{attribute addProperty BoxType "EK1122-0000-0018"}
{attribute addProperty Id "Beckhoff_EJ3xxxsub_EK1100EK1100_179A0949162"}
{attribute addProperty CRC "1763837838"}
{attribute addProperty SizeInBites "16"}
{attribute addProperty SizeInBytes "2"}
TYPE Beckhoff_EJ3xxxEK1122_6922078E EXTENDS EK1122_179A0949 :
STRUCT
	{attribute addProperty Name "Beckhoff_EJ3xxxsub_EK1100"}
	Beckhoff_EJ3xxxsub_EK1100 : EK1100_179A0949;
END_STRUCT
END_TYPE

(* stored: Version 1.2.0.0, ProductVersion 3.1.4024.9
   DUT Beckhoff_EJ3xxxEK1122_6922078E: Id {dbd36f8e-73b1-4117-8fd6-bb816d728d71} *)
